TYPE ST_ListOfVariables_Auhofcenter :
STRUCT
	bIsString				: BOOL;
	sVariableName			: STRING(15);
	sVariableValue			: STRING(30);
END_STRUCT
END_TYPE

(* stored: Version 1.1.0.1, ProductVersion 3.1.4024.9
   DUT ST_ListOfVariables_Auhofcenter: Id {d083cadf-c46f-4647-9b0e-cace6a5b0a20} *)
